{attribute 'strict'}
TYPE E_CSVDataExchangerSelectRowState :
(
	CSV_DATA_EXCHANGER_SELECT_ROW_OPEN_FILE 			:= 0,
	CSV_DATA_EXCHANGER_SELECT_ROW_WAIT_FOR_OPENING		:= 10,	
	CSV_DATA_EXCHANGER_SELECT_ROW_READ_SINGLE_LINE 		:= 20,	
	CSV_DATA_EXCHANGER_SELECT_ROW_WAIT_FOR_READING		:= 30,	
	CSV_DATA_EXCHANGER_SELECT_ROW_PARSE_SINGLE_LINE		:= 40,	
	CSV_DATA_EXCHANGER_SELECT_ROW_CLOSE_FILE			:= 50,	
	CSV_DATA_EXCHANGER_SELECT_ROW_WAIT_FOR_CLOSING		:= 60,
	CSV_DATA_EXCHANGER_SELECT_ROW_READING_DONE			:= 70
);
END_TYPE

(* stored: Version 1.1.0.1, ProductVersion 3.1.4024.9
   DUT E_CSVDataExchangerSelectRowState: Id {02b0d97f-2511-4dbd-bd7c-a20f7f228719} *)
